// TIA Portal V20 export
ORGANIZATION_BLOCK "UpdataVGageDataOB"   // OB10000, LAD, ProgramCycle
TITLE = "Main Program Sweep (Cycle)"
{ S7_Optimized_Access := 'TRUE' }
// stored: AutoNumber false, IsIECCheckEnabled true, SetENOAutomatically false
   VAR_INPUT
      Initial_Call : Bool;   // Initial call of this OB
      Remanence : Bool;   // =True, if remanent data are available
   END_VAR
BEGIN

REGION Network 1 (SCL): Relations Recive Mapping
   // Relations Recive Mapping
   IF "QDAS_InterfaceRelation".Q_DAS.commands.trigger THEN
       "QDAS_ReceiveBuffer".processData := "QDAS_ReceiveRelation".processData;
       "QDAS_ReceiveBuffer".spareOut_1 := "QDAS_ReceiveRelation".spareOut_1;
       "QDAS_ReceiveBuffer".spareOut_2 := "QDAS_ReceiveRelation".spareOut_2;
       "QDAS_ReceiveBuffer".spareOut_3 := "QDAS_ReceiveRelation".spareOut_3;
       "QDAS_ReceiveBuffer".spareOut_4 := "QDAS_ReceiveRelation".spareOut_4;
       "QDAS_ReceiveBuffer".spareOut_5 := "QDAS_ReceiveRelation".spareOut_5;
       "QDAS_ReceiveBuffer".spareOut_6 := "QDAS_ReceiveRelation".spareOut_6;
       "QDAS_ReceiveBuffer".spareOut_7 := "QDAS_ReceiveRelation".spareOut_7;
       "QDAS_ReceiveBuffer".type := "QDAS_ReceiveRelation".type;
       "QDAS_ReceiveBuffer".module := "QDAS_ReceiveRelation".module;
       "QDAS_ReceiveBuffer".machine := "QDAS_ReceiveRelation".machine;
       "QDAS_ReceiveBuffer".fixture := "QDAS_ReceiveRelation".fixture;
       "QDAS_ReceiveBuffer".pun := "QDAS_ReceiveRelation".pun;
       "QDAS_ReceiveBuffer".unWinderInfeed := "QDAS_ReceiveRelation".unWinderInfeed;
       "QDAS_ReceiveBuffer".reelCutInspection := "QDAS_ReceiveRelation".reelCutInspection;
   END_IF;
END_REGION

REGION Network 2: Call QDASDataManager
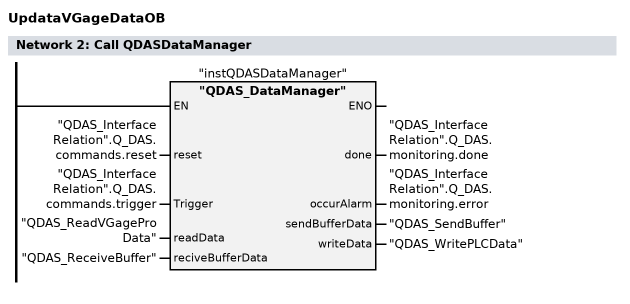
   RUNG wire#powerrail
      "instQDASDataManager"(reset := "QDAS_InterfaceRelation".Q_DAS.commands.reset, Trigger := "QDAS_InterfaceRelation".Q_DAS.commands.trigger, readData := "QDAS_ReadVGageProData", reciveBufferData := "QDAS_ReceiveBuffer", done => "QDAS_InterfaceRelation".Q_DAS.monitoring.done, occurAlarm => "QDAS_InterfaceRelation".Q_DAS.monitoring.error, sendBufferData => "QDAS_SendBuffer", writeData => "QDAS_WritePLCData")
   END_RUNG
   // the same network as SCL:
   "instQDASDataManager"(reset := "QDAS_InterfaceRelation".Q_DAS.commands.reset,   // "QDAS_DataManager"
                         Trigger := "QDAS_InterfaceRelation".Q_DAS.commands.trigger,
                         readData := "QDAS_ReadVGageProData",
                         reciveBufferData := "QDAS_ReceiveBuffer",
                         done => "QDAS_InterfaceRelation".Q_DAS.monitoring.done,
                         occurAlarm => "QDAS_InterfaceRelation".Q_DAS.monitoring.error,
                         sendBufferData => "QDAS_SendBuffer",
                         writeData => "QDAS_WritePLCData");
END_REGION

REGION Network 3 (SCL): Relations Send Mapping
   // Relations Send Mapping
   "QDAS_SendRelation".heartbeatActive := "QDAS_SendBuffer".heartbeatActive;
   "QDAS_SendRelation".dataCollected := "QDAS_SendBuffer".dataCollected;
   "QDAS_SendRelation".plcOK := "QDAS_SendBuffer".plcOK;
   "QDAS_SendRelation".spareIn_1 := "QDAS_SendBuffer".spareIn_1;
   "QDAS_SendRelation".spareIn_2 := "QDAS_SendBuffer".spareIn_2;
   "QDAS_SendRelation".spareIn_3 := "QDAS_SendBuffer".spareIn_3;
   "QDAS_SendRelation".spareIn_4 := "QDAS_SendBuffer".spareIn_4;
   "QDAS_SendRelation".spareIn_5 := "QDAS_SendBuffer".spareIn_5;
END_REGION
END_ORGANIZATION_BLOCK
